(* IEC 61131-3 sources: plc_generation_empirical_study/datasets/task_bank_lean_runtime_v0_1/tasks/C04_R17_lean_composite, 2 files *)

(* ---- interface.st ---- *)
FUNCTION_BLOCK C04_R17_lean_composite
VAR_INPUT
    A_Button : BOOL;
    A_Enable : BOOL;
    A_Reset : BOOL;
    B_ChA : BOOL;
    B_ChB : BOOL;
    B_TestMode : BOOL;
    B_TestPermit : BOOL;
    B_ProcessRequest : BOOL;
    SubsystemBEnable : BOOL;
    CrossReset : BOOL;
END_VAR
VAR_OUTPUT
    A_State : BOOL;
    A_AcceptedPulse : BOOL;
    B_SafeEnable : BOOL;
    B_Disagree : BOOL;
    B_TestActive : BOOL;
    CrossReady : BOOL;
    CrossBlocked : BOOL;
END_VAR
END_FUNCTION_BLOCK

(* ---- reference.st ---- *)
FUNCTION_BLOCK C04_R17_lean_composite
VAR_INPUT
    A_Button : BOOL;
    A_Enable : BOOL;
    A_Reset : BOOL;
    B_ChA : BOOL;
    B_ChB : BOOL;
    B_TestMode : BOOL;
    B_TestPermit : BOOL;
    B_ProcessRequest : BOOL;
    SubsystemBEnable : BOOL;
    CrossReset : BOOL;
END_VAR
VAR_OUTPUT
    A_State : BOOL;
    A_AcceptedPulse : BOOL;
    B_SafeEnable : BOOL;
    B_Disagree : BOOL;
    B_TestActive : BOOL;
    CrossReady : BOOL;
    CrossBlocked : BOOL;
END_VAR
VAR
    A_PrevButton : BOOL := FALSE;
END_VAR

A_AcceptedPulse := FALSE;
IF A_Reset THEN
    A_State := FALSE;
ELSIF A_Enable AND A_Button AND (NOT A_PrevButton) THEN
    A_State := NOT A_State;
    A_AcceptedPulse := TRUE;
END_IF;
A_PrevButton := A_Button;

IF CrossReset THEN
    CrossReady := FALSE;
ELSIF A_State THEN
    CrossReady := TRUE;
END_IF;
CrossBlocked := SubsystemBEnable AND (NOT CrossReady);

IF SubsystemBEnable AND CrossReady THEN
    B_Disagree := B_ChA <> B_ChB;
    B_TestActive := B_TestMode AND B_TestPermit;
    IF B_TestMode THEN
        B_SafeEnable := B_ProcessRequest AND B_TestPermit AND B_ChA;
    ELSE
        B_SafeEnable := B_ProcessRequest AND B_ChA AND B_ChB;
    END_IF;
ELSE
    B_SafeEnable := FALSE;
    B_Disagree := FALSE;
    B_TestActive := FALSE;
END_IF;

END_FUNCTION_BLOCK
